TYPE T_OnlineChangeTestReport :
STRUCT
	bAllRequiredPassed: BOOL;
	bRequiredFailure: BOOL;
	bJsonReady: BOOL;
	bJsonCopyOk: BOOL;
	nJsonLength: UDINT;
	sJson: STRING(2048);
END_STRUCT
END_TYPE

(* stored: Version 1.1.0.1
   DUT T_OnlineChangeTestReport: Id {7ad89472-d072-441d-b4d6-d6f90db311a4} *)
